FUNCTION_BLOCK FB_OPCUA_WorkOnNode_Test  EXTENDS TcUnit.FB_TestSuite
VAR_INPUT
END_VAR
VAR_OUTPUT
END_VAR
VAR
	read	 				: FB_UAreadMock_BoolChangesToTrue;
	write					: FB_UAwriteMock_SetBoolTrue;
	nodeReleaseHandle		: FB_UAnodeReleaseHandleMock_Success;
	nodeGetHandle			: FB_UAnodeGetHandleMock_Success;

	readNode 				: FB_OPCUA_WorkOnNode(
													iOPCUA_Write := write,			
													iOPCUA_Read	:= read,				
													iOPCUA_NodeReleaseHandle := nodeReleaseHandle,	
													iOPCUA_NodeGetHandle :=  nodeGetHandle		
													);
	opcUAreadList_BOOL: ST_OPCUA_NodeVariablePair_BOOL := (clientvariable := booleanToRead, 
															serverNodeIdentifier := 'booleantoread',
															clientVariableInfo := __VARINFO(opcUAreadList_BOOL));
	booleanToRead : BOOL;
	booleanInfo : __SYSTEM.VAR_INFO := __VARINFO(readNode);
END_VAR

variableShouldGetUpdatedWhenChanged();

METHOD variableShouldGetUpdatedWhenChanged
VAR
	sessionCOnnectInfo 		: ST_UASessionConnectInfo;
END_VAR
TEST('variableShouldGetUpdatedWhenChanged');
	
	
	readNode.read(clientVariable := booleanToRead,
					clientVariableAddress := ADR(booleanToRead),
					serverNodeIdentifier := 'test',
					nameSpaceLocationIdentifierEx := 'test',
					ConnectionHdl := 11,
					nNamespaceIndex := 11);
	IF NOT readNode.busy THEN
		assertEquals_BOOL(Expected := TRUE, Actual := booleanToRead, Message := 'Value not updated when changed');
		TEST_FINISHED();
	END_IF
END_METHOD

END_FUNCTION_BLOCK

(* stored: Version 1.1.0.1, ProductVersion 3.1.4024.9
   POU FB_OPCUA_WorkOnNode_Test: Id {f8275c91-08d9-4097-85fd-969f90b067cf}, SpecialFunc None
   Method variableShouldGetUpdatedWhenChanged: Id {fd3e4813-86ce-4fb4-9c27-b1d9ea091390} *)
